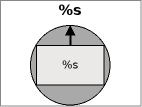
VISUALIZATION VISU_Tube_Rotator  // 142x107
VAR_IN_OUT
    stationName : STRING;
	name : STRING;
    rotAngle : LREAL;
END_VAR
    Ellipse (30,25 80x80)
    Polygon (65,35) (70,25) (75,35)
        p2858320360: rotAngle
    Rectangle (36,45 68x40), "%s", text variable: name
        p2858320360: rotAngle
    Polyline (70,30) (70,45)
        p2858320360: rotAngle
    Rectangle (0,0 140x20), "%s", text variable: stationName
END_VISUALIZATION

(* stored: Version 1.1.0.1, ProductVersion 3.1.4019.2
   Visu VISU_Tube_Rotator: Id {ff4e6d44-c062-4a82-9fb0-d7ff0f10119d} *)
